FUNCTION_BLOCK Mc3PowerTask EXTENDS Mc3MotionTask IMPLEMENTS I_Mc3MotionPowerTask
VAR
	McPower : Tc3_Mc3Ptp.MC_Power;
	{attribute 'hide'}
	_InhibitFeedForward : BOOL;
	{attribute 'hide'}
	_InhibitFeedBackward : BOOL;
END_VAR

{attribute 'monitoring' := 'call'}
PROPERTY Busy : BOOL
GET
Busy := FALSE; (*MC Power Busy behaves busy as long as enabled*)
END_GET
END_PROPERTY

METHOD CyclicLogic
McPower(Axis		   := _Axis.Axis,
		EnablePositive := NOT _InhibitFeedForward,
		EnableNegative := NOT _InhibitFeedBackward,
		Status		   =>,
		Error		   =>,
		ErrorId		   =>);
END_METHOD

METHOD Disable
McPower(Axis		   := _Axis.Axis,
		Enable		   := FALSE,
		EnablePositive := NOT _InhibitFeedForward,
		EnableNegative := NOT _InhibitFeedBackward,
		Status		   =>,
		Error		   =>,
		ErrorId		   =>);
END_METHOD

METHOD Enable
McPower(Axis		   := _Axis.Axis,
		Enable		   := TRUE,
		EnablePositive := NOT _InhibitFeedForward,
		EnableNegative := NOT _InhibitFeedBackward,
		Status		   =>,
		Error		   =>,
		ErrorId		   =>);
END_METHOD

{attribute 'monitoring' := 'call'}
PROPERTY Enabled : BOOL
GET
Enabled := McPower.Status;
END_GET
END_PROPERTY

{attribute 'monitoring' := 'call'}
PROPERTY Error : BOOL
GET
Error := McPower.Error;
END_GET
END_PROPERTY

{attribute 'monitoring' := 'call'}
PROPERTY ErrorId : UDINT
GET
ErrorId := McPower.ErrorID;
END_GET
END_PROPERTY

METHOD Execute : BOOL
Execute := TRUE;
END_METHOD

{attribute 'monitoring' := 'call'}
PROPERTY InhibitFeedBackward : BOOL
GET
InhibitFeedBackward := _InhibitFeedBackward;
END_GET
SET
_InhibitFeedBackward := InhibitFeedBackward;
END_SET
END_PROPERTY

{attribute 'monitoring' := 'call'}
PROPERTY InhibitFeedForward : BOOL
GET
InhibitFeedForward := _InhibitFeedForward;
END_GET
SET
_InhibitFeedForward := InhibitFeedForward;
END_SET
END_PROPERTY

END_FUNCTION_BLOCK

(* stored: Version 1.1.0.1, ProductVersion 3.1.4026.20
   POU Mc3PowerTask: Id {528aff7d-2ac2-4059-9be3-84ea8b07a33b}, SpecialFunc None
   Property Busy: Id {67d24c38-7f44-4500-ba47-3e92a4f494e0}
   Get Get: Id {f49604cb-2fef-4ca3-afbf-5f0b809e9ae8}
   Method CyclicLogic: Id {45ec0260-008f-41a0-b1cb-855471040b1c}
   Method Disable: Id {425b6077-39b7-4e3f-87bf-15c1e2cf7794}
   Method Enable: Id {cf3b7966-332c-4c90-9e1d-37b45483782d}
   Property Enabled: Id {cb81a41b-c7d8-4f97-a340-988ac93abe86}
   Get Get: Id {d806f328-4cc0-4ade-90e6-346575177d89}
   Property Error: Id {dff57e68-d286-4291-83fc-63a983822675}
   Get Get: Id {586025c6-adc2-472f-b3f8-634c662a2018}
   Property ErrorId: Id {f68ef8b5-37a0-484a-bbba-63bf3473a40c}
   Get Get: Id {486de060-3292-4a93-ac2a-df1e9a983680}
   Method Execute: Id {94401452-db2b-46f4-8663-2c7aa986b368}
   Property InhibitFeedBackward: Id {0b9124cf-68de-42e8-bd02-f769409f1730}
   Get Get: Id {86a9d4dd-4801-4204-9244-2aee4991ff99}
   Set Set: Id {d68227af-54d5-44cf-aa6d-153c0cc9744c}
   Property InhibitFeedForward: Id {4e0c2982-5d87-4221-867e-869425609ab3}
   Get Get: Id {4774d7f1-b4c4-462b-a3ef-13bc98f983ca}
   Set Set: Id {b08605c7-2264-4daa-b7b9-738ff5a4dde0} *)
